# EPICS StreamDevice protocol: rsfsxApp/Db/rsfsv.proto
#---------------------------------------------------------------------
# Title      : Rohde & Schwarz FSL Spectrum Analyzer Epics Protocol File
# Project    :
#---------------------------------------------------------------------
# File       : rsfsv.proto
# Author     : Leticia Garcez Capovilla
# Company    : Brazilian Synchrotron Light Laboratory, LNLS/CNPEM
# Created    : 2018-03-19
# Last update: 2019-02-04
#---------------------------------------------------------------------
# Description:
#
# Defines protocol to use the device as a StreamDevice IOC in EPICS
#
#---------------------------------------------------------------------
# Copyright (c) 2018 Brazilian Synchrotron Light Laboratory, LNLS/CNPEM
#
# This program is free software: you can redistribute it and/or
# modify it under the terms of the GNU Lesser General Public License
# as published by the Free Software Foundation, either version 3 of
# the License, or (at your option) any later version.
#
# This program is distributed in the hope that it will be useful, but
# WITHOUT ANY WARRANTY; without even the implied warranty of
# MERCHANTABILITY or FITNESS FOR A PARTICULAR PURPOSE.  See the GNU
# Lesser General Public License for more details.
#
# You should have received a copy of the GNU Lesser General Public
# License along with this program. If not, see
# <http://www.gnu.org/licenses/>.
#---------------------------------------------------------------------
# Revisions  :
# Date        	Version  	Author          	Description
# 2018-mar-19	1.0      	leticiagcapovilla       Created
# 2019-feb-04	2.0		leticiagcapovilla	Updated
#---------------------------------------------------------------------

######################################################################
#
# Variable declaration
#
GLOBAL_TIMEOUT = 5000;

######################################################################
#
# Communication setup
#
OutTerminator = CR LF;
InTerminator = LF;
ExtraInput = Ignore;
MaxInput = 576018;
WriteTimeout = ${GLOBAL_TIMEOUT};
ReadTimeout = ${GLOBAL_TIMEOUT};
ReplyTimeout = ${GLOBAL_TIMEOUT};
Separator = ",";

######################################################################
# Auto Adjust Frequency Scale
#
outAutoFreq {
    out "%{|ADJ:FREQ}";
}

######################################################################
# Auto Adjust Level Scale
#
outAutoLvl {
    out "%{|ADJ:LEV}";
}

######################################################################
# Auto Adjust Frequency and Level Scale
#
outAutoAll {
    out "%{|ADJ:ALL}";
}

######################################################################
# Select Filter Type

inFiltType {
    out "SENS:BWID:RES:TYPE?";
    in "%s";
}

outFiltType {
    out "SENS:BWID:RES:TYPE %{NORM|CFIL|RRC|P5}";
}

######################################################################
# Resolution Bandwidth

inRbw {
    out "SENS:BWID:RES?";
    in "%i";
}

outRbw {
    out "SENS:BWID:RES %s";
}
